Staubli VAL3: onF8Event.pgx

program onF8Event()
  local num l_nSpeedScale
  local num l_nJogVelocity
begin
  // look if the bButton is enable
  if bButton[7]
    // increase the move

    ////    io:direction_pos=true
    ////    wait(getKey()==-1)
    ////    io:direction_pos=false

//    if ! isPowered()
//       call use:timerDialog("请给手臂上电",1)
//      return
//    endIf
//

    if aioGet(MbAI_bMotorPowe)==1
      //7轴正向移动速度
      l_nJogVelocity=100
      ////
      aioSet(MbAO_aJogVelo,l_nJogVelocity)
      aioSet(MbAO_bMoveDir,1)
      aioSet(MbAO_b7Axis,1)
      call use:timerDialog("7轴正向移动...",0)
    else

      if aioGet(MbAI_bMotorPowe)==0
         call use:timerDialog("7轴未上电",1)
        return
      endIf
    endIf

    //
  endIf
end
